PROGRAM P_Demo_FB_DMXGetSensorDefinition
VAR
    fbGetSensorDef    : FB_DMXGetSensorDefinition;    // 读传感器定义
    stDmxCmdBuffer    : ST_DMXCommandBuffer;          // 与通讯 FB 共用
    wTargetManufId    : WORD := 16#4241;              // 目标灯具厂商 ID
    dwTargetDeviceId  : DWORD := 16#12131415;         // 目标灯具设备 ID
    byTargetPort      : BYTE := 0;                    // 根设备通道 0
    bySensorIndex     : BYTE := 0;                    // 第一个传感器
    bDoRead           : BOOL := FALSE;                // 在线给一次上升沿触发
    bBusy             : BOOL;
    bError            : BOOL;
    udiErrId          : UDINT;
    stSensorDef       : ST_DMXSensorDefinition;       // 传感器定义结构
END_VAR

// ============================================================
// Tc2_DMX.FB_DMXGetSensorDefinition 演示程序
// ============================================================
// 场景：把灯具内置温度传感器接入监控：先读传感器定义拿单位(摄氏度)和量程，HMI 才能正确显示。
// 价值：把传感器单位与量程从设备读出，使读数自带物理含义，免去为每个型号硬编码换算系数。
// 验证：设 bySensorIndex:=0，给 bDoRead 一次上升沿 -> bBusy 短暂 TRUE -> 回 FALSE 后 stSensorDef 含该传感器类型/单位/量程；编号越界则 bError 且 udiErrId=0x801B。
// 验证步骤：
//   1. 右键 PLC 项目下 POUs 文件夹 → Add → Existing Item → 选本 .TcPOU 文件
//   2. 引用 Tc2_DMX；同项目里放一个 FB_EL6851CommunicationEx 实例并共用 stDmxCmdBuffer（非 CycleMode）
//   3. 编译 → 登录 → 运行；按上方『验证』行在线给上升沿观察
// ============================================================

fbGetSensorDef(
    bStart                     := bDoRead,
    wDestinationManufacturerId := wTargetManufId,
    dwDestinationDeviceId      := dwTargetDeviceId,
    byPortId                   := byTargetPort,
    bySensorNumber             := bySensorIndex,
    dwOptions                  := 0,
    stCommandBuffer            := stDmxCmdBuffer,
    bBusy                      => bBusy,
    bError                     => bError,
    udiErrorId                 => udiErrId,
    stSensorDefinition         => stSensorDef
);

END_PROGRAM

(* stored: Version 1.1.0.1, ProductVersion 3.1.4024.5
   POU P_Demo_FB_DMXGetSensorDefinition: Id {a25fa889-0331-5afa-90d2-530feeaf3da9}, SpecialFunc None *)
